FUNCTION_BLOCK fb_toggleVal
VAR_INPUT
	IN: BOOL;
END_VAR
VAR_OUTPUT
END_VAR
VAR
END_VAR

IF IN = TRUE AND TCin.ProxUp THEN
	TCout.valvepush := TRUE;
	TCout.valvepull := FALSE;
ELSIF IN = TRUE AND not TCin.ProxUp THEN
	TCout.valvepull := TRUE;
	TCout.valvepush := FALSE;
END_IF

(*
IF IN = TRUE AND TCin.ProxUp THEN
	TCout.valve := FALSE;
ELSIF IN = TRUE AND TCin.ProxDwn THEN
	TCout.valve := TRUE;
END_IF*)

END_FUNCTION_BLOCK

(* stored: Version 1.1.0.1, ProductVersion 3.1.4024.5
   POU fb_toggleVal: Id {1c1b06d7-6701-4c33-a16d-cce0c0c76527}, SpecialFunc None *)
